FUNCTION_BLOCK ServoControl
VAR_INPUT
	bExecute:BOOL;
END_VAR
VAR_OUTPUT
	bDone:BOOL:=FALSE;
	Order:ARRAY[0..7] OF INT:=[2,3,4,5,6,7,8,1];
	CurrentAngle:REAL;
END_VAR
VAR
	ServoBlock:BOOL:=FALSE;
	MoveStart:BOOL:=FALSE;
	MoveFinish:BOOL:=TRUE;
	initAngle:REAL:=0;
	Step:REAL:=-45;
	AnglePush:REAL;
	
	//StatePull:BOOL:=FALSE;
	Angles:ARRAY[0..7] OF REAL:=[0.0,0.0,0.0,0.0,90.0,180.0,180.0,90.0];
	temp:REAL;
	temp_order:INT;
	//该模块第一次运行为到达原点
END_VAR

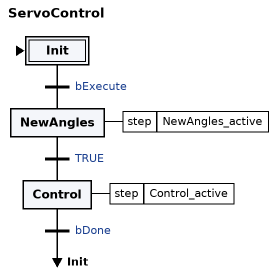
INITIAL_STEP Init:
END_STEP
TRANSITION FROM Init TO NewAngles
    := bExecute;
END_TRANSITION
STEP NewAngles:
    NewAngles_active(N);  // step action
END_STEP
TRANSITION FROM NewAngles TO Control
    := TRUE;
END_TRANSITION
STEP Control:
    Control_active(N);  // step action
END_STEP
TRANSITION FROM Control TO Init
    := bDone;
END_TRANSITION

ACTION Control_active:
IF NOT ServoBlock THEN
	
	//StatePull:=FALSE;
	MoveStart:=TRUE;
	bDone:=MoveFinish;
	IF bDone = TRUE THEN
		MoveStart:=FALSE;
		IF initAngle < -359 THEN
			initAngle:= 0;
		END_IF
		initAngle:=initAngle+Step;
		MoveFinish:=FALSE;
	END_IF
END_IF
END_ACTION

ACTION NewAngles_active:
IF NOT ServoBlock THEN
	temp:=Angles[0];
	Angles[0]:=Angles[1];
	Angles[1]:=Angles[2];
	Angles[2]:=Angles[3];
	Angles[3]:=Angles[4];
	Angles[4]:=Angles[5];
	Angles[5]:=Angles[6];
	Angles[6]:=Angles[7];
	Angles[7]:=temp;
	//Order in world frame
	temp_order:=Order[7];
	Order[7]:=Order[6];
	Order[6]:=Order[5];
	Order[5]:=Order[4];
	Order[4]:=Order[3];
	Order[3]:=Order[2];
	Order[2]:=Order[1];
	Order[1]:=Order[0];
	Order[0]:=temp_order;
	
	AnglePush:=initAngle;
	bDone:=FALSE;
END_IF
END_ACTION

END_FUNCTION_BLOCK

(* stored: Version 1.1.0.1, ProductVersion 3.1.4024.12
   POU ServoControl: Id {14d35239-20af-4930-a088-11bd622831b2}, SpecialFunc None
   Action Control_active: Id {ebd6722f-6b29-4513-8382-eab123f9601e}
   Action NewAngles_active: Id {e7838a9c-4a1c-4a59-9b37-6aeb0494efa3} *)
